# B&R Automation Studio project Parker_BMM_ST_V5_3147_V12 (part 13)

#### pullbottom.c
```c
/********************************************************************
 * COPYRIGHT --  B&R
 ********************************************************************
 * Program: bullbottom
 * File: pullbottom.c
 * Author: lijianjun
 * Created: March 06, 2013
 ********************************************************************
 * Implementation of program coolpin --- pull bottom control
 ********************************************************************/

#include <bur/plctypes.h>

#ifdef _DEFAULT_INCLUDES
	#include <AsDefault.h>
#endif

/**************************************************************************************
                            Function Declarations
**************************************************************************************/

void PullBottom( Mold_typ * pMold);

/**************************************************************************************
     	        		I N I T U P  O F   T H E   T A S K
**************************************************************************************/
_INIT void init ( void )
 {
	LMold.PullBottom.Step = 0;
 	RMold.PullBottom.Step = 0;
 } /* end of _INIT */

 /*************************************************************************************
        				C Y C L I C   P A R T   O F   T H E   T A S K
**************************************************************************************/

 _CYCLIC void cyclic ( void )
 {

	PullBottom(&LMold);
	PullBottom(&RMold);

	gMachineOut.LMold.PullBottom = LMold.ValveOut.PullBottom;
	gMachineOut.RMold.PullBottom = RMold.ValveOut.PullBottom;

 } /* end of _CYCLIC */

void PullBottom( Mold_typ * pMold)
{
   if(0 == pMold->TimeSet.CoolPinUpAlarmTime)pMold->TimeSet.CoolPinUpAlarmTime = 500;

   switch ( pMold->PullBottom.Step )
   {
         /*------------------ stop all the output ------------------*/
         case 0:
            pMold->ValveOut.PullBottom  = 0;
            pMold->ActInfo.PullBottom   = 0;
			pMold->PullBottom.Timer.IN	   = 0;
            break;

      	/*------------------ PullBottom -------------------- */
         case 100: /* PullBottom delay*/
            if(pMold->Option.PullBottom)
            {
				if(pMold->TimeSet.PullBottomDelay != 0)
				{
					pMold->PullBottom.Timer.IN = 1;
					pMold->PullBottom.Timer.PT = pMold->TimeSet.PullBottomDelay;
					pMold->PullBottom.Step = 200;
				}
				else
				{
					pMold->PullBottom.Step = 300;
				}

            }
            else
            {
            	pMold->PullBottom.Step = 900;
            }
          	break;

         case 200: /* delay ok */
            pMold->TimeDis.PullBottomDelay = pMold->PullBottom.Timer.ET;
            if (1 == pMold->PullBottom.Timer.Q)
            {
               pMold->PullBottom.Timer.IN       = 0;
               pMold->TimeDis.CoolPinDnDelay = 0;
               pMold->PullBottom.Step = 300;
            }
            break;

         case 300:

            if(pMold->TimeSet.PullBottomTime != 0)
            {
               pMold->PullBottom.Timer.IN = 1;
               pMold->PullBottom.Timer.PT = pMold->TimeSet.PullBottomTime;
               pMold->PullBottom.Step = 400;
            }
            else
            {
               pMold->PullBottom.Step = 500;
            }
            break;

         case 400: /*PullBottom time*/
            pMold->ActInfo.PullBottom  = 1;
            pMold->ValveOut.PullBottom = 1;

            pMold->TimeDis.PullBottomTime = pMold->PullBottom.Timer.ET;
            if (1 == pMold->PullBottom.Timer.Q)
            {
               pMold->ValveOut.PullBottom = 0;
               pMold->PullBottom.Timer.IN = 0;
//               pMold->TimeDis.PullBottomTime = 0;
               pMold->PullBottom.Step = 500;
            }

            break;

		case 500:
			pMold->ActInfo.PullBottom  = 0;
			pMold->ValveOut.PullBottom = 0;

			pMold->PullBottom.Step = 900;

			break;

         case 900:

			pMold->ActInfo.PullBottom  = 0;
			pMold->ValveOut.PullBottom = 0;

			pMold->PullBottom.Timer.IN = 0;

			pMold->PullBottom.Step = 3000;

            break;

		case 1100:      /* bCoolPinUpNextCycClampCls  autorun Case-4570 */
						/* 強制桿下到下一循環關模後才轉一上 */

			pMold->ActInfo.CoolPinDn  = 1;
			pMold->ValveOut.CoolPinDn = 1;

			break;

         case 3000:
            break;

		case 5000:
			pMold->ActInfo.PullBottom  = 1;
			pMold->ValveOut.PullBottom = 1;

			break;

         case 20000:
            pMold->ActInfo.PullBottom  = 0;
            pMold->ValveOut.PullBottom = 0;

			pMold->PullBottom.Timer.IN = 0;
            pMold->PullBottom.Step = 0;
            break;

		case 30000:
			pMold->ActInfo.PullBottom  = 0;
			pMold->ValveOut.PullBottom = 0;

			pMold->PullBottom.Timer.IN = 0;
			pMold->PullBottom.Step = 0;
            break;

   }/* end of switch */

	/* ----------------- pull bottom  action limit --------------------  */
	if(pMold->PullBottom.Step > 100 && pMold->PullBottom.Step < 900)
	{

	}

}/*end of function */
```

### Program Logical/process/hookpin (ANSIC, version 1.00.0) - hook pin

#### hookpin.c
```c
/********************************************************************
 * COPYRIGHT --  B&R
 ********************************************************************
 * Program: HookPin
 * File: HookPin.c
 * Author: lijianjun
 * Created: March 06, 2013
 ********************************************************************
 * Implementation of program HookPin --- cooling pin control
 ********************************************************************/

#include <bur/plctypes.h>

#ifdef _DEFAULT_INCLUDES
#include <AsDefault.h>
#endif

/**************************************************************************************
                            Function Declarations
**************************************************************************************/

void HookPin( Mold_typ * pMold);

/**************************************************************************************
     	        		I N I T U P  O F   T H E   T A S K
**************************************************************************************/
_INIT void init ( void )
{
	LMold.HookPin.Step = 0;
	RMold.HookPin.Step = 0;
} /* end of _INIT */

 /*************************************************************************************
        				C Y C L I C   P A R T   O F   T H E   T A S K
**************************************************************************************/

_CYCLIC void cyclic ( void )
{

	LMold.TransDIn.HookPinFwLimit = gMachineIn.LMold.HookPinFwLimit;
	RMold.TransDIn.HookPinFwLimit = gMachineIn.RMold.HookPinFwLimit;

	LMold.TransDIn.HookPinBwLimit = gMachineIn.LMold.HookPinBwLimit;
	RMold.TransDIn.HookPinBwLimit = gMachineIn.RMold.HookPinBwLimit;

	HookPin(&LMold);
	HookPin(&RMold);

	gMachineOut.LMold.HookPinFw = LMold.ValveOut.HookPinFw;
	gMachineOut.RMold.HookPinFw = RMold.ValveOut.HookPinFw;

} /* end of _CYCLIC */

void HookPin( Mold_typ * pMold)
{
	if(0 == pMold->TimeSet.HookPinFwAlarmTime)pMold->TimeSet.HookPinFwAlarmTime = 500;
	if(0 == pMold->TimeSet.HookPinBwAlarmTime)pMold->TimeSet.HookPinBwAlarmTime = 500;

	switch ( pMold->HookPin.Step )
	{
		/*------------------ stop all the output ------------------*/
		case 0:
//			pMold->ActInfo.HookPinFw   = 0;
//			pMold->ValveOut.HookPinFw  = 0;

			pMold->HookPin.LimitTimer.IN	   = 0;
			pMold->HookPin.Timer.IN	   = 0;
			break;

		/*--------------------------------------------------- */
		/*---------------- HookPin Fw  --------------------- */
		/*--------------------------------------------------- */
		case 100: /* HookPin delay*/
			if(pMold->Option.HookPin)
			{
				if(pMold->TimeSet.HookPinFwDelay != 0)
				{
					pMold->HookPin.Timer.IN = 1;
					pMold->HookPin.Timer.PT = pMold->TimeSet.HookPinFwDelay;
					pMold->HookPin.Step = 200;
				}
				else
				{
					pMold->HookPin.Step = 300;
				}
			}
			else
			{
				pMold->HookPin.Step = 300;
			}
			break;

		case 200: /* delay ok */
			pMold->TimeDis.HookPinFwDelay = pMold->HookPin.Timer.ET;
			if (1 == pMold->HookPin.Timer.Q)
			{
				pMold->HookPin.Timer.IN       = 0;
				//               pMold->TimeDis.HookPinFwDelay = 0;
				pMold->HookPin.Step = 300;
			}
			break;

		case 300:
			if(pMold->Option.HookPin)
			{
				pMold->HookPin.LimitTimer.IN = 1;
				pMold->HookPin.LimitTimer.PT = pMold->TimeSet.HookPinFwAlarmTime;
				pMold->HookPin.Step = 400;
			}
			else
			{
				pMold->HookPin.Step = 2900;  // for no use
			}

			break;

		case 400:
			pMold->ActInfo.HookPinFw  = 1;
			pMold->ValveOut.HookPinFw = 1;

			if (1 == pMold->TransDIn.HookPinFwLimit)
			{
				pMold->HookPin.Step = 500;
			}

			break;

		case 500:

			pMold->HookPin.LimitTimer.IN	   = 0;
			pMold->HookPin.Timer.IN	   = 0;

			pMold->HookPin.Step = 3000;
			break;

		case 2900:  // for no use

			pMold->ActInfo.HookPinFw   = 0;
			pMold->ValveOut.HookPinFw  = 0;

			pMold->HookPin.LimitTimer.IN	   = 0;
			pMold->HookPin.Timer.IN	   = 0;

			pMold->HookPin.Step = 3000;

			break;

		case 3000:
			break;

		case 5000:
			pMold->ActInfo.HookPinFw  = 1;
			pMold->ValveOut.HookPinFw = 1;

			break;

		/*--------------------------------------------------- */
		/*---------------- HookPin Bw  --------------------- */
		/*--------------------------------------------------- */

		case 10100: /* HookPin delay*/
			if(pMold->Option.HookPin)
			{
				if(pMold->TimeSet.HookPinBwDelay != 0)
				{
					pMold->HookPin.Timer.IN = 1;
					pMold->HookPin.Timer.PT = pMold->TimeSet.HookPinBwDelay;
					pMold->HookPin.Step = 10200;
				}
				else
				{
					pMold->HookPin.Step = 10300;
				}
			}
			else
			{
				pMold->HookPin.Step = 10300;
			}
			break;

		case 10200: /* delay ok */
			pMold->TimeDis.HookPinBwDelay = pMold->HookPin.Timer.ET;
			if (1 == pMold->HookPin.Timer.Q)
			{
				pMold->HookPin.Timer.IN       = 0;
				//               pMold->TimeDis.HookPinFwDelay = 0;
				pMold->HookPin.Step = 10300;
			}
			break;

		case 10300:

			if(pMold->Option.HookPin)
			{
				pMold->HookPin.LimitTimer.IN = 1;
				pMold->HookPin.LimitTimer.PT = pMold->TimeSet.HookPinBwAlarmTime;
				pMold->HookPin.Step = 10400;
			}
			else
			{

				if (1 == pMold->TransDIn.HookPinBwLimit)
				{
					pMold->HookPin.Step = 12900;  // for no use
				}
				else
				{
					pMold->Alarm.HookPinNotAtBwPos = 1;
					pMold->HookPin.Step = 40000;           /*  HookPin bw alarm   */
				}
			}

			break;

		case 10400:

			pMold->ActInfo.HookPinFw  = 0;
			pMold->ValveOut.HookPinFw = 0;

			if (1 == pMold->TransDIn.HookPinBwLimit)
			{
				pMold->HookPin.Step = 10500;
			}

			break;

		case 10500:

			pMold->ActInfo.HookPinFw   = 0;
			//			pMold->ValveOut.HookPinFw  = 0;

			pMold->HookPin.LimitTimer.IN	   = 0;
			pMold->HookPin.Timer.IN	   = 0;

			pMold->HookPin.Step = 13000;

			break;

		case 12900:  // for no use

			pMold->ActInfo.HookPinFw   = 0;
			pMold->ValveOut.HookPinFw  = 0;

			pMold->HookPin.LimitTimer.IN	   = 0;
			pMold->HookPin.Timer.IN	   = 0;

			pMold->HookPin.Step = 13000;

			break;

		case 13000:

			break;

		case 15000:
			pMold->ActInfo.HookPinFw  = 0;
			pMold->ValveOut.HookPinFw = 0;

			break;

		case 20000:
//			pMold->ActInfo.HookPinFw   = 0;
//			pMold->ValveOut.HookPinFw  = 0;

			pMold->HookPin.LimitTimer.IN	   = 0;
			pMold->HookPin.Timer.IN	   = 0;

			pMold->HookPin.Step	   = 0;
			break;

		case 30000:
			//			pMold->ActInfo.HookPinFw   = 0;
			//			pMold->ValveOut.HookPinFw  = 0;

			pMold->HookPin.LimitTimer.IN	   = 0;
			pMold->HookPin.Timer.IN	   = 0;

			pMold->HookPin.Step	   = 0;
			break;

		case 40000:
			//			pMold->ActInfo.HookPinFw   = 0;
			//			pMold->ValveOut.HookPinFw  = 0;

			pMold->HookPin.LimitTimer.IN	   = 0;
			pMold->HookPin.Timer.IN	   = 0;

			break;

		case 41000:
			//			pMold->ActInfo.HookPinFw   = 0;
			//			pMold->ValveOut.HookPinFw  = 0;

			pMold->HookPin.LimitTimer.IN	   = 0;
			pMold->HookPin.Timer.IN	   = 0;

			pMold->HookPin.Step	   = 40000;

			break;
	}/* end of switch */

	/* ----------------- HookPin Fw / Bw timeout --------------------  */
	if(1 == pMold->HookPin.LimitTimer.Q && 1 == gMachineInfo.TimeLimit)
	{
		if(pMold->HookPin.Step < 500 && pMold->HookPin.Step > 300)		/* HookPin Fw  */
		{
			pMold->Alarm.HookPinNotAtFwPos = 1;
		}

		if(pMold->TopDeflash.Step < 10500 && pMold->TopDeflash.Step > 10300)	/* HookPin Bw  */
		{
			pMold->Alarm.HookPinNotAtBwPos = 1;
		}

		pMold->HookPin.Step = 41000;
	}

	/* ----------------- Angle pin Fw  action limit --------------------  */
	if(pMold->HookPin.Step > 300 && pMold->HookPin.Step < 500)
	{
		if( 0 == pMold->Carriage.BwPos )
		{
			pMold->Alarm.CarriageNotAtBwDI= 1;
			pMold->HookPin.Step = 40000;
		}
	}

}/*end of function */
```

### Program Logical/process/coolpin (ANSIC, version 1.00.0) - cool pin

#### coolpin.c
```c
/********************************************************************
 * COPYRIGHT --  B&R
 ********************************************************************
 * Program: coolpin
 * File: coolpin.c
 * Author: lijianjun
 * Created: March 06, 2013
 ********************************************************************
 * Implementation of program coolpin --- cooling pin control
 ********************************************************************/

#include <bur/plctypes.h>

#ifdef _DEFAULT_INCLUDES
#include <AsDefault.h>
#endif

/**************************************************************************************
                            Function Declarations
**************************************************************************************/

void CoolPin( Mold_typ * pMold);

/**************************************************************************************
     	        		I N I T U P  O F   T H E   T A S K
**************************************************************************************/
_INIT void init ( void )
{
	LMold.CoolPin.Step = 0;
	RMold.CoolPin.Step = 0;
} /* end of _INIT */

 /*************************************************************************************
        				C Y C L I C   P A R T   O F   T H E   T A S K
**************************************************************************************/

_CYCLIC void cyclic ( void )
{

	LMold.TransDIn.CoolPinUpLimit = gMachineIn.LMold.CoolPinUpLimit;
	RMold.TransDIn.CoolPinUpLimit = gMachineIn.RMold.CoolPinUpLimit;

	CoolPin(&LMold);
	CoolPin(&RMold);

	gMachineOut.LMold.CoolPinDn = LMold.ValveOut.CoolPinDn;
	gMachineOut.RMold.CoolPinDn = RMold.ValveOut.CoolPinDn;

} /* end of _CYCLIC */

void CoolPin( Mold_typ * pMold)
{
	if(0 == pMold->TimeSet.CoolPinUpAlarmTime)pMold->TimeSet.CoolPinUpAlarmTime = 500;

	switch ( pMold->CoolPin.Step )
	{
		/*------------------ stop all the output ------------------*/
		case 0:
//			pMold->ValveOut.CoolPinDn  = 0;
//			pMold->ActInfo.CoolPinDn   = 0;
			pMold->CoolPin.LimitTimer.IN	   = 0;
			pMold->CoolPin.Timer.IN	   = 0;
			break;

		/*------------------ CoolPin -------------------- */
		case 100: /* CoolPin delay*/
			if(pMold->Option.CoolPin)
			{
				if ( 1 == gMachineFix.Option.bCoolPinUpNextCycClampCls)    /*  於下一循環關模後轉一上    */
				{
					pMold->CoolPin.Step = 1100; 		/*  強制桿下到下一循環關模後才轉一上 */
				}
				else
				{
					if(pMold->TimeSet.CoolPinDnDelay != 0)
					{
						pMold->CoolPin.Timer.IN = 1;
						pMold->CoolPin.Timer.PT = pMold->TimeSet.CoolPinDnDelay;
						pMold->CoolPin.Step = 200;

						//gExSPC
						if(pMold == & LMold)
						{
							gExSPC[ExIndex].LMold.CoolPinDnDelay = pMold->TimeSet.CoolPinDnDelay/100.0;
						}
						else
						{
							gExSPC[ExIndex].RMold.CoolPinDnDelay = pMold->TimeSet.CoolPinDnDelay/100.0;
						}
					}
					else
					{
						pMold->CoolPin.Step = 300;
					}
				}
			}
			else
			{
				pMold->CoolPin.Step = 900;
			}
			break;

		case 200: /* delay ok */
			pMold->TimeDis.CoolPinDnDelay = pMold->CoolPin.Timer.ET;
			if (1 == pMold->CoolPin.Timer.Q)
			{
				pMold->CoolPin.Timer.IN       = 0;
				//               pMold->TimeDis.CoolPinDnDelay = 0;
				pMold->CoolPin.Step = 300;
			}
			break;

		case 300: //沒有轉一下時間， 轉一下直到轉一吹冷結束

			//            if(pMold->TimeSet.CoolPinDnTime != 0)
			//            {
			//               pMold->CoolPin.Timer.IN = 1;
			//               pMold->CoolPin.Timer.PT = pMold->TimeSet.CoolPinDnTime;
			//               pMold->CoolPin.Step = 400;
			//
			//				//gExSPC
			//				if(pMold == & LMold)
			//				{
			//					gExSPC[ExIndex].LMold.CoolPinDnTime = pMold->TimeSet.CoolPinDnTime/100.0;
			//				}
			//				else
			//				{
			//					gExSPC[ExIndex].RMold.CoolPinDnTime = pMold->TimeSet.CoolPinDnTime/100.0;
			//				}
			//            }
			//            else
			//            {
			//               pMold->CoolPin.Step = 500;
			//            }

			pMold->CoolPin.Step = 400;
			break;

		case 400:
			pMold->ActInfo.CoolPinDn  = 1;
			pMold->ValveOut.CoolPinDn = 1;

			//            pMold->TimeDis.CoolPinDnTime = pMold->CoolPin.Timer.ET;
			//            if (1 == pMold->CoolPin.Timer.Q)
			//            {
			//               pMold->ValveOut.CoolPinDn = 0;
			//               pMold->CoolPin.Timer.IN = 0;
			//               pMold->TimeDis.CoolPinDnTime = 0;
			//               pMold->CoolPin.Step = 500;
			//            }

			if (3000==pMold->CoolPinBlow.Step)
			{
				pMold->CoolPin.Step = 500;
			}

			break;

		case 500:

			if ((1 == pMold->Option.CoolPin) || (1 == pMold->ValveOut.CoolPinDn))
			{
				pMold->CoolPin.LimitTimer.IN = 1;
				pMold->CoolPin.LimitTimer.PT = pMold->TimeSet.CoolPinUpAlarmTime;
				pMold->CoolPin.Step = 600;
			}
			else
			{
				pMold->CoolPin.Step = 650;	// for no use
			}

			break;

		case 600:
			pMold->ActInfo.CoolPinDn  = 0;
			pMold->ValveOut.CoolPinDn = 0;

			if(pMold->TransDIn.CoolPinUpLimit)
			{
				pMold->CoolPin.Step = 900;
			}
			pMold->TimeDis.CoolPinUpAlarmTime = pMold->CoolPin.LimitTimer.ET;
			if (1 == pMold->CoolPin.LimitTimer.Q)
			{
				pMold->ActInfo.CoolPinDn  = 0;
				pMold->ValveOut.CoolPinDn = 0;

				pMold->CoolPin.LimitTimer.IN = 0;
				pMold->Alarm.CoolPinNotAtUpPos = 1;

				pMold->CoolPin.Step = 40000;
			}
			break;

		case 650: // for no use
			//			pMold->ActInfo.CoolPinDn  = 0;
			//			pMold->ValveOut.CoolPinDn = 0;

			if(pMold->TransDIn.CoolPinUpLimit)
			{
				pMold->CoolPin.Step = 900;
			}
			else
			{
				pMold->CoolPin.LimitTimer.IN = 0;
				pMold->Alarm.CoolPinNotAtUpPos = 1;

				pMold->CoolPin.Step = 40000;
			}

			//			pMold->TimeDis.CoolPinUpAlarmTime = pMold->CoolPin.LimitTimer.ET;
			//			if (1 == pMold->CoolPin.LimitTimer.Q)
			//			{
			//				pMold->CoolPin.LimitTimer.IN = 0;
			//				pMold->Alarm.CoolPinNotAtUpPos = 1;
			//
			//				pMold->CoolPin.Step = 40000;
			//			}
			break;

		case 900:

			pMold->ValveOut.CoolPinDn = 0;
			pMold->ActInfo.CoolPinDn  = 0;
			pMold->CoolPin.LimitTimer.IN = 0;
			pMold->CoolPin.Step = 3000;
			break;

		case 1100:      /* bCoolPinUpNextCycClampCls  autorun Case-4570 */
			/* 強制桿下到下一循環關模後才轉一上 */

			pMold->ActInfo.CoolPinDn  = 1;
			pMold->ValveOut.CoolPinDn = 1;

			break;

		case 3000:
			break;

		case 5000:
			pMold->ActInfo.CoolPinDn  = 1;
			pMold->ValveOut.CoolPinDn = 1;

			break;

		case 15000:
			pMold->ActInfo.CoolPinDn  = 0;
			pMold->ValveOut.CoolPinDn = 0;

			break;

		case 20000:
//			pMold->ActInfo.CoolPinDn  = 0;
//			pMold->ValveOut.CoolPinDn = 0;

			pMold->CoolPin.Timer.IN = 0;
			pMold->CoolPin.LimitTimer.IN = 0;
			pMold->CoolPin.Step = 0;
			break;

		case 30000:
//			pMold->ActInfo.CoolPinDn  = 0;
//			pMold->ValveOut.CoolPinDn = 0;
			pMold->CoolPin.Timer.IN = 0;
			pMold->CoolPin.LimitTimer.IN = 0;
			pMold->CoolPin.Step = 0;
			break;

		case 40000:
//			pMold->ActInfo.CoolPinDn  = 0;
//			pMold->ValveOut.CoolPinDn = 0;
			pMold->CoolPin.Timer.IN = 0;
			pMold->CoolPin.LimitTimer.IN = 0;

			break;
	}/* end of switch */

	/* ----------------- cool pin down  action limit --------------------  */
	if(pMold->CoolPin.Step > 100 && pMold->CoolPin.Step < 900)
	{

	}

}/*end of function */
```

### Program Logical/process/coolpin2 (ANSIC, version 1.00.0) - cool pin 2

#### coolpin2.c
```c
/********************************************************************
 * COPYRIGHT --  B&R
 ********************************************************************
 * Program: coolpin2
 * File: coolpin2.c
 * Author: lijianjun
 * Created: March 06, 2013
 ********************************************************************
 * Implementation of program coolpin2 --- cooling pin 2 control
 ********************************************************************/

#include <bur/plctypes.h>

#ifdef _DEFAULT_INCLUDES
	#include <AsDefault.h>
#endif

/**************************************************************************************
                            Function Declarations
**************************************************************************************/

void CoolPin2( Mold_typ * pMold);

/**************************************************************************************
     	        		I N I T U P  O F   T H E   T A S K
**************************************************************************************/
_INIT void init ( void )
 {
 	LMold.CoolPin2.Step = 0;
 	RMold.CoolPin2.Step = 0;
 } /* end of _INIT */

 /*************************************************************************************
        				C Y C L I C   P A R T   O F   T H E   T A S K
**************************************************************************************/

 _CYCLIC void cyclic ( void )
 {
 	LMold.TransDIn.CoolPin2UpLimit = gMachineIn.LMold.CoolPin2UpLimit;
 	RMold.TransDIn.CoolPin2UpLimit = gMachineIn.RMold.CoolPin2UpLimit;

	CoolPin2(&LMold);
	CoolPin2(&RMold);

	gMachineOut.LMold.CoolPin2Dn = LMold.ValveOut.CoolPin2Dn;
	gMachineOut.RMold.CoolPin2Dn = RMold.ValveOut.CoolPin2Dn;

 } /* end of _CYCLIC */

void CoolPin2( Mold_typ * pMold)
{
	if(0 == pMold->TimeSet.CoolPin2UpAlarmTime)pMold->TimeSet.CoolPin2UpAlarmTime = 500;

	switch ( pMold->CoolPin2.Step )
	{
		/*------------------ stop all the output ------------------*/
		case 0:
//			pMold->CoolPin2.Out   	   = 0;
//			pMold->ValveOut.CoolPin2Dn  = 0;
//			pMold->ActInfo.CoolPin2Dn   = 0;
			pMold->CoolPin2.Timer.IN	   = 0;
			pMold->CoolPin2.LimitTimer.IN	   = 0;
			break;

		/*------------------ CoolPin2 -------------------- */
		case 100: /* CoolPin2 delay*/
			if(pMold->Option.CoolPin2)
			{
				if(pMold->TimeSet.CoolPin2DnDelay != 0)
				{
					pMold->CoolPin2.Timer.IN = 1;
					pMold->CoolPin2.Timer.PT = pMold->TimeSet.CoolPin2DnDelay;
					pMold->CoolPin2.Step = 200;
				}
				else
				{
					pMold->CoolPin2.Step = 300;
				}
			}
			else
			{
				pMold->CoolPin2.Step = 500;
			}

			break;
		case 200: /* delay ok */
			pMold->TimeDis.CoolPin2DnDelay = pMold->CoolPin2.Timer.ET;
			if (1 == pMold->CoolPin2.Timer.Q)
			{
				pMold->CoolPin2.Timer.IN       = 0;
				//		pMold->TimeDis.CoolPin2DnDelay = 0;
				pMold->CoolPin2.Step = 400;
			}
			break;

		case 300:  //沒有轉二下時間， 轉二下直到轉二吹冷結束
			//            	if(pMold->TimeSet.CoolPin2DnTime != 0)
			//            	{
			//            		pMold->CoolPin2.Timer.IN = 1;
			//					pMold->CoolPin2.Timer.PT = pMold->TimeSet.CoolPin2DnTime;
			//					pMold->CoolPin2.Step = 400;
			//            	}
			//            	else
			//            	{
			//            		pMold->CoolPin2.Step = 500;
			//            	}
			pMold->CoolPin2.Step = 400;
			break;

		case 400:
			pMold->ActInfo.CoolPin2Dn  = 1;
			pMold->ValveOut.CoolPin2Dn = 1;
			pMold->CoolPin2.Out        = 1;

			//            	pMold->TimeDis.CoolPin2DnTime = pMold->CoolPin2.Timer.ET;
			//            	if (1 == pMold->CoolPin2.Timer.Q)
			//            	{
			//            		pMold->CoolPin2.Out        = 0;
			//            		pMold->ValveOut.CoolPin2Dn = 0;
			//            		pMold->CoolPin2.Timer.IN = 0;
			//            		pMold->TimeDis.CoolPin2DnTime = 0;
			//            		pMold->CoolPin2.Step = 500;
			//            	}
			if (3000==pMold->CoolPin2Blow.Step)
			{
				pMold->CoolPin2.Step = 500;
			}

			break;

		case 500:
			pMold->CoolPin2.Timer.IN = 0;
			pMold->CoolPin2.Step = 550;
			break;

		case 550:
			if (1 == pMold->Option.CoolPin2)
			{
				pMold->CoolPin2.LimitTimer.IN = 1;
				pMold->CoolPin2.LimitTimer.PT = pMold->TimeSet.CoolPin2UpAlarmTime;
				pMold->CoolPin2.Step = 600;
			}
			else
			{
				pMold->CoolPin2.Step = 650;	// for no use
			}

			break;

		case 600:
			pMold->ActInfo.CoolPin2Dn  = 0;
			pMold->CoolPin2.Out        = 0;
			pMold->ValveOut.CoolPin2Dn = 0;

			if(1 == pMold->TransDIn.CoolPin2UpLimit)
			{
				pMold->CoolPin2.Step = 900;
			}
			pMold->TimeDis.CoolPin2UpAlarmTime = pMold->CoolPin2.LimitTimer.ET;

			if (1 == pMold->CoolPin2.LimitTimer.Q)
			{
				pMold->ActInfo.CoolPin2Dn  = 0;
				pMold->CoolPin2.Out        = 0;
				pMold->ValveOut.CoolPin2Dn = 0;

				pMold->CoolPin2.LimitTimer.IN = 0;
				pMold->Alarm.CoolPin2NotAtUpPos = 1;

				pMold->CoolPin2.Step = 40000;
			}
			break;

		case 650: // for no use

			if(pMold->TransDIn.CoolPin2UpLimit)
			{
				pMold->CoolPin2.Step = 900;
			}
			else
			{
				pMold->CoolPin2.LimitTimer.IN = 0;
				pMold->Alarm.CoolPin2NotAtUpPos = 1;
				pMold->CoolPin2.Step = 40000;
			}

			//			pMold->TimeDis.CoolPin2UpAlarmTime = pMold->CoolPin2.Timer.ET;
			//			if (1 == pMold->CoolPin2.Timer.Q)
			//			{
			//			//	pMold->ActInfo.CoolPin2Dn  = 0;
			//			//	pMold->CoolPin2.Out        = 0;
			//			//	pMold->ValveOut.CoolPin2Dn = 0;
			//
			//				pMold->CoolPin2.Timer.IN = 0;
			//				pMold->Alarm.CoolPin2NotAtUpPos = 1;
			//
			//				pMold->CoolPin2.Step = 40000;
			//			}
			break;

		case 900:
			if (1==gMachineInfo.Auto)
			{
				if(pMold == &RMold)
				{
					RMold.Option.CoolPin2 = gMacOption.RCoolPin2;
				}
				else
				{
					LMold.Option.CoolPin2 = gMacOption.LCoolPin2;
				}
			}
			pMold->CoolPin2.Out      = 0;
			pMold->ValveOut.CoolPin2Dn  = 0;
			pMold->ActInfo.CoolPin2Dn   = 0;

			pMold->CoolPin2.Timer.IN = 0;
			pMold->CoolPin2.LimitTimer.IN = 0;
			pMold->CoolPin2.Step = 3000;
			break;
		case 3000:

			break;

		case 5000:
			pMold->ActInfo.CoolPin2Dn  = 1;
			pMold->ValveOut.CoolPin2Dn = 1;

			break;

		case 15000:
			pMold->ActInfo.CoolPin2Dn  = 0;
			pMold->ValveOut.CoolPin2Dn = 0;

			break;

		case 20000:
//			pMold->CoolPin2.Out        = 0;
//			pMold->ActInfo.CoolPin2Dn  = 0;
//			pMold->ValveOut.CoolPin2Dn = 0;

			pMold->CoolPin2.Timer.IN = 0;
			pMold->CoolPin2.LimitTimer.IN = 0;
			pMold->CoolPin2.Step    = 0;
			break;

		case 30000:
//			pMold->CoolPin2.Out        = 0;
//			pMold->ActInfo.CoolPin2Dn  = 0;
//			pMold->ValveOut.CoolPin2Dn = 0;
			pMold->CoolPin2.Timer.IN = 0;
			pMold->CoolPin2.LimitTimer.IN = 0;
			pMold->CoolPin2.Step     = 0;
			break;

		case 40000:
//			pMold->CoolPin2.Out        = 0;
//			pMold->ActInfo.CoolPin2Dn  = 0;
//			pMold->ValveOut.CoolPin2Dn = 0;
			pMold->CoolPin2.Timer.IN = 0;
			pMold->CoolPin2.LimitTimer.IN = 0;

			break;

		case 41000:
			//			pMold->CoolPin2.Out        = 0;
			//			pMold->ActInfo.CoolPin2Dn  = 0;
			//			pMold->ValveOut.CoolPin2Dn = 0;
			pMold->CoolPin2.Timer.IN = 0;
			pMold->CoolPin2.LimitTimer.IN = 0;
			pMold->CoolPin2.Step     = 40000;
			break;

	}/* end of switch */

	/* ----------------- cool pin2 down  action limit --------------------  */
	if(pMold->CoolPin2.Step > 100 && pMold->CoolPin2.Step < 900)
	{

	}

}/*end of function */
```

### Program Logical/process/coolpin3 (ANSIC, version 1.00.0) - cool pin 3

#### coolpin3.c
```c
/********************************************************************
 * COPYRIGHT --  B&R
 ********************************************************************
 * Program: coolpin3
 * File: coolpin3.c
 * Author: lijianjun
 * Created: March 06, 2013
 ********************************************************************
 * Implementation of program coolpin3 --- cooling pin 3 control
 ********************************************************************/

#include <bur/plctypes.h>

#ifdef _DEFAULT_INCLUDES
#include <AsDefault.h>
#endif

/**************************************************************************************
                            Function Declarations
**************************************************************************************/

void CoolPin3( Mold_typ * pMold);

/**************************************************************************************
     	        		I N I T U P  O F   T H E   T A S K
**************************************************************************************/
_INIT void init ( void )
{
	LMold.CoolPin3.Step = 0;
	RMold.CoolPin3.Step = 0;
} /* end of _INIT */

 /*************************************************************************************
        				C Y C L I C   P A R T   O F   T H E   T A S K
**************************************************************************************/

_CYCLIC void cyclic ( void )
{
	LMold.TransDIn.CoolPin3UpLimit = gMachineIn.LMold.CoolPin3UpLimit;
	RMold.TransDIn.CoolPin3UpLimit = gMachineIn.RMold.CoolPin3UpLimit;

	CoolPin3(&LMold);
	CoolPin3(&RMold);

	gMachineOut.LMold.CoolPin3Dn = LMold.ValveOut.CoolPin3Dn;
	gMachineOut.RMold.CoolPin3Dn = RMold.ValveOut.CoolPin3Dn;

} /* end of _CYCLIC */

void CoolPin3( Mold_typ * pMold)
{

	if(0 == pMold->TimeSet.CoolPin3UpAlarmTime)pMold->TimeSet.CoolPin3UpAlarmTime = 500;

	switch ( pMold->CoolPin3.Step )
	{
		/*------------------ stop all the output ------------------*/
		case 0:
//			pMold->ActInfo.CoolPin3Dn   = 0;
//			pMold->ValveOut.CoolPin3Dn  = 0;

			pMold->CoolPin3.LimitTimer.IN = 0;
			pMold->CoolPin3.Timer.IN	= 0;
			break;

		/*------------------ CoolPin3 -------------------- */
		case 100: /* CoolPin3 delay*/
			if(pMold->Option.CoolPin3)
			{
				if(pMold->TimeSet.CoolPin3DnDelay != 0)
				{
					pMold->CoolPin3.Timer.IN = 1;
					pMold->CoolPin3.Timer.PT = pMold->TimeSet.CoolPin3DnDelay;
					pMold->CoolPin3.Step = 200;
				}
				else
				{
					pMold->CoolPin3.Step = 400;
				}
			}
			else
			{
				pMold->CoolPin3.Step = 900;
			}
			break;
		case 200: /* delay ok */
			pMold->TimeDis.CoolPin3DnDelay = pMold->CoolPin3.Timer.ET;
			if (1 == pMold->CoolPin3.Timer.Q)
			{
				pMold->CoolPin3.Timer.IN       = 0;
				//	pMold->TimeDis.CoolPin3DnDelay = 0;
				pMold->CoolPin3.Step = 400;
			}
			break;
		case 300:  //沒有轉三下時間， 轉三下直到轉三吹冷結束
			//            	if(pMold->TimeSet.CoolPin3DnTime != 0)
			//            	{
			//            		pMold->CoolPin3.Timer.IN = 1;
			//					pMold->CoolPin3.Timer.PT = pMold->TimeSet.CoolPin3DnTime;
			//					pMold->CoolPin3.Step = 400;
			//            	}
			//            	else
			//            	{
			//            		pMold->CoolPin3.Step = 500;
			//            	}
			pMold->CoolPin3.Step = 400;

			break;
		case 400:
			pMold->ActInfo.CoolPin3Dn  = 1;
			pMold->ValveOut.CoolPin3Dn = 1;

			//            	pMold->TimeDis.CoolPin3DnTime = pMold->CoolPin3.Timer.ET;
			//            	if (1 == pMold->CoolPin3.Timer.Q)
			//            	{
			//            		pMold->ValveOut.CoolPin3Dn = 0;
			//            		pMold->CoolPin3.Timer.IN = 0;
			//            		pMold->TimeDis.CoolPin3DnTime = 0;
			//            		pMold->CoolPin3.Step = 450;
			//            	}
			if (3000==pMold->CoolPin3Blow.Step)
			{
				pMold->CoolPin3.Step = 500;
			}
			break;

		case 500:
			pMold->CoolPin3.Timer.IN = 0;
			pMold->CoolPin3.Step = 550;

			break;

		case 550:
			if (1 == pMold->Option.CoolPin3)
			{
				pMold->CoolPin3.LimitTimer.IN = 1;
				pMold->CoolPin3.LimitTimer.PT = pMold->TimeSet.CoolPin3UpAlarmTime;
				pMold->CoolPin3.Step = 600;
			}
			else
			{
				pMold->CoolPin3.Step = 650;	// for no use
			}

			break;

		case 600:
			pMold->ActInfo.CoolPin3Dn  = 0;
			pMold->ValveOut.CoolPin3Dn = 0;

			if(pMold->TransDIn.CoolPin3UpLimit)
			{
				pMold->CoolPin3.Step = 900;
			}
			pMold->TimeDis.CoolPin3UpAlarmTime = pMold->CoolPin3.LimitTimer.ET;
			if (1 == pMold->CoolPin3.LimitTimer.Q)
			{
				pMold->ActInfo.CoolPin3Dn  = 0;
				pMold->ValveOut.CoolPin3Dn = 0;

				pMold->CoolPin3.LimitTimer.IN = 0;
				pMold->Alarm.CoolPin3NotAtUpPos = 1;

				pMold->CoolPin3.Step = 40000;
			}
			break;

		case 650: // for no use

			if(pMold->TransDIn.CoolPin3UpLimit)
			{
				pMold->CoolPin3.Step = 900;
			}
			else
			{
				pMold->CoolPin3.LimitTimer.IN = 0;
				pMold->Alarm.CoolPin3NotAtUpPos = 1;
				pMold->CoolPin3.Step = 40000;
			}

			break;

		case 900:
			if (1==gMachineInfo.Auto)
			{
				if(pMold == &RMold)
				{
					RMold.Option.CoolPin3 = gMacOption.RCoolPin3;
				}
				else
				{
					LMold.Option.CoolPin3 = gMacOption.LCoolPin3;
				}
			}

			pMold->ValveOut.CoolPin3Dn  = 0;
			pMold->ActInfo.CoolPin3Dn   = 0;

			pMold->CoolPin3.Timer.IN = 0;
			pMold->CoolPin3.LimitTimer.IN = 0;
			pMold->CoolPin3.Step = 3000;

			break;

		case 3000:

			break;

		case 5000:
			pMold->ActInfo.CoolPin3Dn  = 1;
			pMold->ValveOut.CoolPin3Dn = 1;

			break;

		case 15000:
			pMold->ActInfo.CoolPin3Dn  = 0;
			pMold->ValveOut.CoolPin3Dn = 0;

			break;

		case 20000:
//			pMold->ActInfo.CoolPin3Dn  = 0;
//			pMold->ValveOut.CoolPin3Dn = 0;

			pMold->CoolPin3.Timer.IN = 0;
			pMold->CoolPin3.LimitTimer.IN = 0;
			pMold->CoolPin3.Step    = 0;
			break;

		case 30000:
//			pMold->ActInfo.CoolPin3Dn  = 0;
//			pMold->ValveOut.CoolPin3Dn = 0;

			pMold->CoolPin3.Timer.IN = 0;
			pMold->CoolPin3.LimitTimer.IN = 0;
			pMold->CoolPin3.Step     = 0;
			break;

		case 40000:
//			pMold->ActInfo.CoolPin3Dn  = 0;
//			pMold->ValveOut.CoolPin3Dn = 0;

			pMold->CoolPin3.Timer.IN = 0;
			pMold->CoolPin3.LimitTimer.IN = 0;

			break;

		case 41000:
			//			pMold->ActInfo.CoolPin3Dn  = 0;
			//			pMold->ValveOut.CoolPin3Dn = 0;

			pMold->CoolPin3.Timer.IN = 0;
			pMold->CoolPin3.LimitTimer.IN = 0;
			pMold->CoolPin3.Step     = 40000;
			break;

	}/* end of switch */

	/* ----------------- cool pin3 down  action limit --------------------  */
	if(pMold->CoolPin3.Step > 100 && pMold->CoolPin3.Step < 900)
	{

	}

}/*end of function */
```

### Program Logical/process/coolblw (ANSIC, version 1.00.0) - cooling blow

#### coolblow.c
```c
/********************************************************************
 * COPYRIGHT --  B&R
 ********************************************************************
 * Program: coolblow
 * File: coolblow.c
 * Author: lijianjun
 * Created: March 06, 2013
 ********************************************************************
 * Implementation of program coolblow --- cooling blow control
 ********************************************************************/

#include <bur/plctypes.h>
#ifdef _DEFAULT_INCLUDES
	#include <AsDefault.h>
#endif

/**************************************************************************************
                            Function Declarations
**************************************************************************************/

void CoolPinBlow( Mold_typ * pMold);

/**************************************************************************************
     	        		I N I T U P  O F   T H E   T A S K
**************************************************************************************/
_INIT void init ( void )
 {
 	LMold.CoolPinBlow.Step = 0;
 	RMold.CoolPinBlow.Step = 0;
 } /* end of _INIT */

 /*************************************************************************************
        				C Y C L I C   P A R T   O F   T H E   T A S K
**************************************************************************************/

 _CYCLIC void cyclic ( void )
 {
	CoolPinBlow(&LMold);
	CoolPinBlow(&RMold);

	gMachineOut.LMold.CoolPinBlow = LMold.ValveOut.CoolPinBlow;
	gMachineOut.RMold.CoolPinBlow = RMold.ValveOut.CoolPinBlow;

 } /* end of _CYCLIC */

void CoolPinBlow( Mold_typ * pMold)
{

	 switch ( pMold->CoolPinBlow.Step )
     {
      		/*------------------ stop all the output ------------------*/
            case 0:
            	pMold->ValveOut.CoolPinBlow   = 0;
            	pMold->ActInfo.CoolPinBlow  = 0;
            	pMold->CoolPinBlow.Timer.IN	= 0;
            	break;

      		/*------------------ CoolPin -------------------- */
            case 100:
            	if(pMold->Option.CoolPin)
      			{
	            	if(pMold->TimeSet.CoolPinBlowDelay != 0)
		      		{
	      				pMold->CoolPinBlow.Timer.IN = 1;
						pMold->CoolPinBlow.Timer.PT = pMold->TimeSet.CoolPinBlowDelay;
	      				pMold->CoolPinBlow.Step = 200;

						//gExSPC
						if(pMold == & LMold)
						{
							gExSPC[ExIndex].LMold.CoolPinBlowDelay = pMold->TimeSet.CoolPinBlowDelay/100.0;
						}
						else
						{
							gExSPC[ExIndex].RMold.CoolPinBlowDelay = pMold->TimeSet.CoolPinBlowDelay/100.0;
						}
	      			}
	      			else
	      			{
	      				pMold->CoolPinBlow.Step = 300;
	      			}
	      		}
	      		else
	      		{
	      			pMold->CoolPinBlow.Step = 900;
	      		}
            	break;
            case 200:
            	pMold->TimeDis.CoolPinBlowDelay = pMold->CoolPinBlow.Timer.ET;
            	if (1 == pMold->CoolPinBlow.Timer.Q)
            	{
            		pMold->CoolPinBlow.Timer.IN       = 0;
            	//	pMold->TimeDis.CoolPinBlowDelay = 0;
            		pMold->CoolPinBlow.Step = 300;
            	}
            	break;
            case 300:
            	if(pMold->TimeSet.CoolPinBlowTime != 0)
            	{
            		pMold->CoolPinBlow.Timer.IN = 1;
					pMold->CoolPinBlow.Timer.PT = pMold->TimeSet.CoolPinBlowTime;
					pMold->CoolPinBlow.Step = 400;

					//gExSPC
					if(pMold == & LMold)
					{
						gExSPC[ExIndex].LMold.CoolPinBlowTime = pMold->TimeSet.CoolPinBlowTime/100.0;
					}
					else
					{
						gExSPC[ExIndex].RMold.CoolPinBlowTime = pMold->TimeSet.CoolPinBlowTime/100.0;
					}

            	}
            	else
            	{
            		pMold->CoolPinBlow.Step = 900;
            	}
            	break;
            case 400:
            	pMold->ActInfo.CoolPinBlow  = 1;
            	pMold->ValveOut.CoolPinBlow = 1;

            	pMold->TimeDis.CoolPinBlowTime = pMold->CoolPinBlow.Timer.ET;
            	if (1 == pMold->CoolPinBlow.Timer.Q)
            	{
            		pMold->CoolPinBlow.Timer.IN = 0;
            	//	pMold->TimeDis.CoolPinBlowTime = 0;

            		pMold->CoolPinBlow.Step = 500;
            	}
            	break;

			case 500:
				pMold->ActInfo.CoolPinBlow  = 0;
				pMold->ValveOut.CoolPinBlow = 0;

				pMold->CoolPinBlow.Step = 900;

				break;

            case 900:
//			if (1==gMachineInfo.Auto)
//			{
//				if(pMold == &RMold)
//				{
//					RMold.Option.CoolPin = gMacOption.RCoolPin;
//				}
//				else
//				{
//					LMold.Option.CoolPin = gMacOption.LCoolPin;
//				}
//			}
            	pMold->ActInfo.CoolPinBlow  = 0;
            	pMold->ValveOut.CoolPinBlow = 0;

            	pMold->CoolPinBlow.Timer.IN = 0;

            	pMold->CoolPinBlow.Step = 3000;
            	break;

            case 3000:
            	break;

			case 5000:
				pMold->ActInfo.CoolPinBlow  = 1;
				pMold->ValveOut.CoolPinBlow = 1;

				break;

            case 20000:
            	pMold->ActInfo.CoolPinBlow  = 0;
            	pMold->ValveOut.CoolPinBlow = 0;

				pMold->CoolPinBlow.Timer.IN = 0;
				pMold->CoolPinBlow.Step    = 0;
				break;

			case 30000:
            	pMold->ActInfo.CoolPinBlow  = 0;
            	pMold->ValveOut.CoolPinBlow = 0;

				pMold->CoolPinBlow.Timer.IN = 0;
				pMold->CoolPinBlow.Step     = 0;
				break;

	 }/* end of switch */

	/* ----------------- cool pin blow  action limit --------------------  */
	 if(pMold->CoolPinBlow.Step > 100 && pMold->CoolPinBlow.Step < 900)
	 {
	 	if( 0 == pMold->Option.CoolPin && 1 == gMachineInfo.Auto)
	 	{
			pMold->CoolPinBlow.Step  = 900;
		}
	}
}/*end of function */
```

### Program Logical/process/coolblw2 (ANSIC, version 1.00.0) - cool blow 2

#### coolblow2.c
```c
/********************************************************************
 * COPYRIGHT --  B&R
 ********************************************************************
 * Program: coolblow
 * File: coolblow.c
 * Author: lijianjun
 * Created: March 06, 2013
 ********************************************************************
 * Implementation of program coolblow --- cooling blow control
 ********************************************************************/

#include <bur/plctypes.h>

#ifdef _DEFAULT_INCLUDES
#include <AsDefault.h>
#endif

/**************************************************************************************
                            Function Declarations
**************************************************************************************/

void CoolPin2Blow( Mold_typ * pMold);

/**************************************************************************************
     	        		I N I T U P  O F   T H E   T A S K
**************************************************************************************/
_INIT void init ( void )
 {
 	LMold.CoolPin2Blow.Step = 0;
 	RMold.CoolPin2Blow.Step = 0;
 } /* end of _INIT */

 /*************************************************************************************
        				C Y C L I C   P A R T   O F   T H E   T A S K
**************************************************************************************/

 _CYCLIC void cyclic ( void )
 {
	CoolPin2Blow(&LMold);
	CoolPin2Blow(&RMold);

	gMachineOut.LMold.CoolPin2Blow = LMold.ValveOut.CoolPin2Blow;
	gMachineOut.RMold.CoolPin2Blow = RMold.ValveOut.CoolPin2Blow;

 } /* end of _CYCLIC */

void CoolPin2Blow( Mold_typ * pMold)
{

	 switch ( pMold->CoolPin2Blow.Step )
     {
      		/*------------------ stop all the output ------------------*/
            case 0:
            	pMold->CoolPin2Blow.Out   	= 0;
            	pMold->ActInfo.CoolPin2Blow  = 0;
            	pMold->CoolPin2Blow.Timer.IN	= 0;
            	break;

      		/*------------------ CoolPin2 -------------------- */
            case 100:
            	if(pMold->Option.CoolPin2)
      			{
	            	if(pMold->TimeSet.CoolPin2BlowDelay != 0)
		      		{
	      				pMold->CoolPin2Blow.Timer.IN = 1;
						pMold->CoolPin2Blow.Timer.PT = pMold->TimeSet.CoolPin2BlowDelay;
	      				pMold->CoolPin2Blow.Step = 200;
	      			}
	      			else
	      			{
	      				pMold->CoolPin2Blow.Step = 300;
	      			}
	      		}
	      		else
	      		{
	      			pMold->CoolPin2Blow.Step = 900;
	      		}
            	break;
            case 200:
            	pMold->TimeDis.CoolPin2BlowDelay = pMold->CoolPin2Blow.Timer.ET;
            	if (1 == pMold->CoolPin2Blow.Timer.Q)
            	{
            		pMold->CoolPin2Blow.Timer.IN       = 0;
            //		pMold->TimeDis.CoolPin2BlowDelay = 0;
            		pMold->CoolPin2Blow.Step = 300;
            	}
            	break;
            case 300:
            	if(pMold->TimeSet.CoolPin2BlowTime != 0)
            	{
            		pMold->CoolPin2Blow.Timer.IN = 1;
					pMold->CoolPin2Blow.Timer.PT = pMold->TimeSet.CoolPin2BlowTime;
					pMold->CoolPin2Blow.Step = 400;
            	}
            	else
            	{
            		pMold->CoolPin2Blow.Step = 900;
            	}
            	break;
            case 400:
            	pMold->CoolPin2Blow.Out      = 1;
            	pMold->ActInfo.CoolPin2Blow  = 1;
            	pMold->ValveOut.CoolPin2Blow = 1;

            	pMold->TimeDis.CoolPin2BlowTime = pMold->CoolPin2Blow.Timer.ET;
            	if (1 == pMold->CoolPin2Blow.Timer.Q)
            	{
            		pMold->CoolPin2Blow.Out      = 0;
            		pMold->ActInfo.CoolPin2Blow  = 0;
            		pMold->ValveOut.CoolPin2Blow = 0;

            		pMold->CoolPin2Blow.Timer.IN = 0;
            	//	pMold->TimeDis.CoolPin2BlowTime = 0;

            		pMold->CoolPin2Blow.Step = 900;
            	}
            	break;
            case 900:
//			if (1==gMachineInfo.Auto)
//			{
//				if(pMold == &RMold)
//				{
//					RMold.Option.CoolPin2 = gMacOption.RCoolPin2;
//				}
//				else
//				{
//					LMold.Option.CoolPin2 = gMacOption.LCoolPin2;
//				}
//			}
            	pMold->CoolPin2Blow.Out      = 0;
            	pMold->ActInfo.CoolPin2Blow  = 0;
            	pMold->ValveOut.CoolPin2Blow = 0;

            	pMold->CoolPin2Blow.Timer.IN = 0;

            	pMold->CoolPin2Blow.Step = 3000;
            	break;

            case 3000:
            	break;

			case 5000:
				pMold->ActInfo.CoolPin2Blow  = 1;
				pMold->ValveOut.CoolPin2Blow = 1;

				break;

            case 20000:
            	pMold->CoolPin2Blow.Out      = 0;
            	pMold->ActInfo.CoolPin2Blow  = 0;
            	pMold->ValveOut.CoolPin2Blow = 0;

				pMold->CoolPin2Blow.Timer.IN = 0;
				pMold->CoolPin2Blow.Step    = 0;
				break;

			case 30000:
            	pMold->CoolPin2Blow.Out      = 0;
            	pMold->ActInfo.CoolPin2Blow  = 0;
            	pMold->ValveOut.CoolPin2Blow = 0;

				pMold->CoolPin2Blow.Timer.IN = 0;
				pMold->CoolPin2Blow.Step     = 0;
				break;

	 }/* end of switch */

	 if(pMold->CoolPin2Blow.Step > 100 && pMold->CoolPin2Blow.Step < 500)
	 {
	 	if(!pMold->Option.CoolPin2 && 1 == gMachineInfo.Auto)
	 	{
			pMold->CoolPin2Blow.Step  = 900;
		}
	}
}/*end of function */
```

### Program Logical/process/coolblw3 (ANSIC, version 1.00.0) - cool blow 3

#### coolblow3.c
```c
/********************************************************************
 * COPYRIGHT --  B&R
 ********************************************************************
 * Program: coolblow
 * File: coolblow.c
 * Author: lijianjun
 * Created: March 06, 2013
 ********************************************************************
 * Implementation of program coolblow --- cooling blow control
 ********************************************************************/

#include <bur/plctypes.h>

#ifdef _DEFAULT_INCLUDES
#include <AsDefault.h>
#endif

/**************************************************************************************
                            Function Declarations
**************************************************************************************/

void CoolPin3Blow( Mold_typ * pMold);

/**************************************************************************************
     	        		I N I T U P  O F   T H E   T A S K
**************************************************************************************/
_INIT void init ( void )
 {
 	LMold.CoolPin3Blow.Step = 0;
 	RMold.CoolPin3Blow.Step = 0;
 } /* end of _INIT */

 /*************************************************************************************
        				C Y C L I C   P A R T   O F   T H E   T A S K
**************************************************************************************/

 _CYCLIC void cyclic ( void )
 {
	CoolPin3Blow(&LMold);
	CoolPin3Blow(&RMold);

	gMachineOut.LMold.CoolPin3Blow = LMold.ValveOut.CoolPin3Blow;
	gMachineOut.RMold.CoolPin3Blow = RMold.ValveOut.CoolPin3Blow;

 } /* end of _CYCLIC */

void CoolPin3Blow( Mold_typ * pMold)
{

	 switch ( pMold->CoolPin3Blow.Step )
     {
      		/*------------------ stop all the output ------------------*/
            case 0:
            	pMold->CoolPin3Blow.Out   	= 0;
            	pMold->ActInfo.CoolPin3Blow  = 0;
            	pMold->CoolPin3Blow.Timer.IN	= 0;
            	break;

      		/*------------------ CoolPin3 -------------------- */
            case 100:
            	if(pMold->Option.CoolPin3)
      			{
	            	if(pMold->TimeSet.CoolPin3BlowDelay != 0)
		      		{
	      				pMold->CoolPin3Blow.Timer.IN = 1;
						pMold->CoolPin3Blow.Timer.PT = pMold->TimeSet.CoolPin3BlowDelay;
	      				pMold->CoolPin3Blow.Step = 200;
	      			}
	      			else
	      			{
	      				pMold->CoolPin3Blow.Step = 300;
	      			}
	      		}
	      		else
	      		{
	      			pMold->CoolPin3Blow.Step = 900;
	      		}
            	break;
            case 200:
            	pMold->TimeDis.CoolPin3BlowDelay = pMold->CoolPin3Blow.Timer.ET;
            	if (1 == pMold->CoolPin3Blow.Timer.Q)
            	{
            		pMold->CoolPin3Blow.Timer.IN       = 0;
            	//	pMold->TimeDis.CoolPin3BlowDelay = 0;
            		pMold->CoolPin3Blow.Step = 300;
            	}
            	break;
            case 300:
            	if(pMold->TimeSet.CoolPin3BlowTime != 0)
            	{
            		pMold->CoolPin3Blow.Timer.IN = 1;
					pMold->CoolPin3Blow.Timer.PT = pMold->TimeSet.CoolPin3BlowTime;
					pMold->CoolPin3Blow.Step = 400;
            	}
            	else
            	{
            		pMold->CoolPin3Blow.Step = 900;
            	}
            	break;
            case 400:
            	pMold->CoolPin3Blow.Out      = 1;
            	pMold->ActInfo.CoolPin3Blow  = 1;
            	pMold->ValveOut.CoolPin3Blow = 1;

            	pMold->TimeDis.CoolPin3BlowTime = pMold->CoolPin3Blow.Timer.ET;
            	if (1 == pMold->CoolPin3Blow.Timer.Q)
            	{
            		pMold->CoolPin3Blow.Out      = 0;
            		pMold->ActInfo.CoolPin3Blow  = 0;
            		pMold->ValveOut.CoolPin3Blow = 0;

            		pMold->CoolPin3Blow.Timer.IN = 0;
            	//	pMold->TimeDis.CoolPin3BlowTime = 0;

            		pMold->CoolPin3Blow.Step = 900;
            	}
            	break;
            case 900:
//			if (1==gMachineInfo.Auto)
//			{
//				if(pMold == &RMold)
//				{
//					RMold.Option.CoolPin3 = gMacOption.RCoolPin3;
//				}
//				else
//				{
//					LMold.Option.CoolPin3 = gMacOption.LCoolPin3;
//				}
//			}
            	pMold->CoolPin3Blow.Out      = 0;
            	pMold->ActInfo.CoolPin3Blow  = 0;
            	pMold->ValveOut.CoolPin3Blow = 0;

            	pMold->CoolPin3Blow.Timer.IN = 0;

            	pMold->CoolPin3Blow.Step = 3000;
            	break;

            case 3000:
            	break;

			case 5000:
				pMold->ActInfo.CoolPin3Blow  = 1;
				pMold->ValveOut.CoolPin3Blow = 1;

				break;

            case 20000:
            	pMold->CoolPin3Blow.Out      = 0;
            	pMold->ActInfo.CoolPin3Blow  = 0;
            	pMold->ValveOut.CoolPin3Blow = 0;

				pMold->CoolPin3Blow.Timer.IN = 0;
				pMold->CoolPin3Blow.Step    = 0;
				break;

			case 30000:
            	pMold->CoolPin3Blow.Out      = 0;
            	pMold->ActInfo.CoolPin3Blow  = 0;
            	pMold->ValveOut.CoolPin3Blow = 0;

				pMold->CoolPin3Blow.Timer.IN = 0;
				pMold->CoolPin3Blow.Step     = 0;
				break;

	 }/* end of switch */

	 if(pMold->CoolPin3Blow.Step > 100 && pMold->CoolPin3Blow.Step < 500)
	 {
	 	if(!pMold->Option.CoolPin3 && 1 == gMachineInfo.Auto)
	 	{
			pMold->CoolPin3Blow.Step  = 900;
		}
	}
}/*end of function */
```

### Program Logical/process/cutter (ANSIC, version 1.00.0) - cutter

#### cutter.c
```c
/********************************************************************
 * COPYRIGHT --  B&R
 ********************************************************************
 * Program: cutter
 * File: cutter.c
 * Author: lijianjun
 * Created: March 06, 2013
 ********************************************************************
 * Implementation of program cutter --- cutter control
 ********************************************************************/

#include <bur/plctypes.h>

#ifdef _DEFAULT_INCLUDES
#include <AsDefault.h>
#endif

#include "edge.h"

/**************************************************************************************
                            Function Declarations
**************************************************************************************/

void Cutter( Mold_typ * pMold);

/**************************************************************************************
     	        		I N I T U P  O F   T H E   T A S K
**************************************************************************************/
_INIT void init ( void )
 {
 	LMold.Cutter.Step = 0;
 	RMold.Cutter.Step = 0;
 } /* end of _INIT */

 /*************************************************************************************
        				C Y C L I C   P A R T   O F   T H E   T A S K
**************************************************************************************/

 _CYCLIC void cyclic ( void )
 {

	Cutter(&LMold);
	Cutter(&RMold);

//	if(1 == gMachineInfo.Auto)
//	{
//		if( 1 == LMold.Option.CutterMode)	/*  双向切刀 */
//		{
//			if(0 == LMold.ValveOut.Cutter && 0 == RMold.ValveOut.Cutter)
//			{
//				gMachineOut.CutterFw = 0;
//				gMachineOut.CutterBw = 0;
//			}
//			else if(1 == LMold.ValveOut.Cutter || 1 == RMold.ValveOut.Cutter)
//			{
//				gMachineOut.CutterFw = 1;
//				gMachineOut.CutterBw = 0;
//			}
//			else
//			{
//				gMachineOut.CutterFw = 0;
//				gMachineOut.CutterBw = 1;
//			}
//		}
//		else								/*  单向切刀 */
//		{
//			if (EDGEPOS(LMold.ValveOut.Cutter ,Cutter_L_P) || EDGEPOS(RMold.ValveOut.Cutter ,Cutter_R_P))
//			{
//				if(0 == gMachineOut.CutterBw)
//				{
//					gMachineOut.CutterFw = !gMachineOut.CutterFw;
//				}
//
//				if(0 == gMachineOut.CutterFw)
//				{
//					gMachineOut.CutterBw = !gMachineOut.CutterBw;
//					if(0 == gMachineOut.CutterBw)gMachineOut.CutterFw = ! gMachineOut.CutterFw;
//				}
//			}
//		}
//	}
//	else
//	{
//		if(0 == LMold.ValveOut.Cutter && 0 == RMold.ValveOut.Cutter)
//		{
//			gMachineOut.CutterFw = 0;
//			gMachineOut.CutterBw = 0;
//		}
//		else if(1 == LMold.ValveOut.Cutter || 1 == RMold.ValveOut.Cutter)
//		{
//			gMachineOut.CutterFw = 1;
//			gMachineOut.CutterBw = 0;
//		}
//		else
//		{
//			gMachineOut.CutterFw = 0;
//			gMachineOut.CutterBw = 1;
//		}
//	}

//	Cutter_L_P = LMold.ValveOut.Cutter;
//	Cutter_R_P = RMold.ValveOut.Cutter;

	gMachineOut.CutterFw = LMold.ValveOut.Cutter | RMold.ValveOut.Cutter;
 } /* end of _CYCLIC */

void Cutter( Mold_typ * pMold)
{
	 switch ( pMold->Cutter.Step )
     {
      		/*------------------ stop all the output ------------------*/
            case 0:
//            	pMold->ValveOut.Cutter  	   = 0;
//            	pMold->ActInfo.Cutter  = 0;

            	pMold->Cutter.Timer.IN	= 0;
            	break;

      		/*------------------ Cutter course -------------------- */
      		case 100: /* close delay*/
			if ( pMold->Option.Cutter)
			{
				if(pMold->TimeSet.CutterDelay != 0)
				{
					pMold->Cutter.Timer.IN = 1;
					pMold->Cutter.Timer.PT = pMold->TimeSet.CutterDelay;
					pMold->Cutter.Step 	   = 200;
				}
				else
				{
					pMold->Cutter.Step = 300;
				}
			}
			else
			{
				pMold->Cutter.Step = 3000;
			}

             	break;

            case 200: /* delay ok */
            	pMold->TimeDis.CutterDelay = pMold->Cutter.Timer.ET;
            	if (1 == pMold->Cutter.Timer.Q)
            	{
            		pMold->Cutter.Timer.IN     = 0;
            	//	pMold->TimeDis.CutterDelay = 0;
            		pMold->Cutter.Step = 300;
            	}
            	break;

            case 300:/*Determine Cutter mode , if double cutter goes to 400, single cutter goes to 1100*/
					/*   涨气启动   */
//				RMold.SupportAir.Step = 100;
				if(1 == gMachineInfo.Auto)
				{
//						if(RMold.SupportAir.Step == 0)RMold.SupportAir.Step = 100;

					if(1 == RMold.Option.Enable && 1 == LMold.Option.Enable)
					{
						if(pMold == &RMold)
						{
							LMold.OnceSupport  = 1;
						}
						else
						{
							RMold.OnceSupport  = 1;
						}
					}
					else
					{
						pMold->OnceSupport  = 1;
					}
				}

            	if( 1 == pMold->Option.CutterMode)/*Double Cutter*/
            	{
					if( 0 ==  pMold->ValveOut.Cutter)
					{
						if( SUPPORTAIR_MODE_STANDARD == gMachineFix.MoldR.SupportAir.eSupportAirMode)
						{
							pMold->SupportAir.Step = 100;// air support， only for double cutter
						}

						if(pMold->TimeSet.CutterTime != 0)
						{
							pMold->Cutter.Timer.IN = 1;
							pMold->Cutter.Timer.PT = pMold->TimeSet.CutterTime;
							pMold->Cutter.Step = 400;
						}
						else
						{
							/*   cutter time gAlarm   */
							pMold->Cutter.Step = 450;
						}

					}
					else /*If cutter is retain on Fw position , then do Single Cutter again to go back Bw Position*/
					{
						pMold->Cutter.Step = 1100;
					}

	            }
	            else/*Single Cutter*/
	            {
	            	pMold->Cutter.Step = 1100;
	            }
            	break;

            case 400:/*Double cutter, move forward until time expired*/
            	pMold->ActInfo.Cutter = 1;
				pMold->ValveOut.Cutter  = 1;

            	pMold->TimeDis.CutterTime = pMold->Cutter.Timer.ET;
            	if (1 == pMold->Cutter.Timer.Q)
            	{
            		pMold->Cutter.Timer.IN    = 0;
            //		pMold->TimeDis.CutterTime = 0;
					pMold->Cutter.Step = 450;/*Change to case 450*/
            	}
            	break;

			case 450:/*Time expire or no cutter time setting*/
				pMold->ValveOut.Cutter = 0;
				pMold->ActInfo.Cutter  = 0;

				pMold->Cutter.Step 	  = 3000;
			break;

            case 500:/*Current no used case*/
            	pMold->Cutter.Timer.IN = 1;
					pMold->Cutter.Timer.PT = pMold->TimeSet.CutterBwTime;
					pMold->Cutter.Step = 600;
            	break;

            case 600:/*Current no used case*/
            	pMold->ValveOut.Cutter     = 2;
            	pMold->ActInfo.Cutter = 1;

            	pMold->TimeDis.CutterBwTime = pMold->Cutter.Timer.ET;
            	if (1 == pMold->Cutter.Timer.Q)
            	{
            		pMold->Cutter.Timer.IN      = 0;
            	//	pMold->TimeDis.CutterBwTime = 0;
            		pMold->Cutter.Step = 700;
            	}
				break;

            case 700:/*Current no used case*/
            	pMold->ValveOut.Cutter = 0;
            	pMold->ActInfo.Cutter  = 0;

				pMold->Cutter.Step = 800;
            	break;

            case 800:/*Current no used case*/
            	pMold->ValveOut.Cutter     = 0;
            	pMold->ActInfo.Cutter = 0;

            	pMold->Cutter.Step = 3000;
            	break;

            case 1100:/*Single cutter , inverse output*/
            	pMold->ValveOut.Cutter = !pMold->ValveOut.Cutter;/*Albert*/
            	pMold->ActInfo.Cutter = pMold->ValveOut.Cutter;
            	pMold->Cutter.Step = 3000;
            	break;

            case 1200:/*Current no used case*/
            	pMold->Cutter.Step = 1300;
            	break;

            case 1300:/*Current no used case*/
               	pMold->ValveOut.Cutter     = 0;
            	pMold->ActInfo.Cutter = 0;

            	pMold->Cutter.Step = 3000;
            	break;

            case 3000:
            	break;

			case 5000:
				pMold->ValveOut.Cutter     = 1;
				pMold->ActInfo.Cutter = 1;
				break;

            /*--------------- Manual action stop -----------------*/
            case 20000:
				if(pMold->Option.CutterMode)/*Albert Double cutter*/
				{
					pMold->ValveOut.Cutter      = 0;
				}

					pMold->Cutter.Timer.IN = 0;

				//	pMold->TimeDis.CutterTime  = 0;
				//	pMold->TimeDis.CutterDelay = 0;

					pMold->ActInfo.Cutter  = 0;
					pMold->Cutter.Step 	   = 0;
					break;

			/*--------------- Instance stop -----------------*/
			case 30000:
				if(pMold->Option.CutterMode)/*Albert Double Cutter*/
				{
					pMold->ValveOut.Cutter      = 0;
				}
				pMold->Cutter.Timer.IN = 0;

			//	pMold->TimeDis.CutterTime  = 0;
			//	pMold->TimeDis.CutterDelay = 0;

				pMold->ActInfo.Cutter  = 0;
				pMold->Cutter.Step     = 0;
				break;

	 }/* end of switch */
}/*end of function */
```

#### cutter.var
```iecst
VAR
	Cutter_R_P	:USINT;
	Cutter_L_P	:USINT;
END_VAR
```

- edge.h (reference to Logical/GlobalIncludes/edge.h)

### Program Logical/process/sensor (ANSIC, version 1.00.0) - sensor up / down

#### sensor.c
```c
/********************************************************************
 * COPYRIGHT --  B&R China
 ********************************************************************
 * Program: Tonnage
 * File: Tonnage.c
 * Author: lijianjun
 * Created: March 06, 2013
 ********************************************************************
 * Implementation of program Tonnage --- mold Tonnage
 ********************************************************************/

#include <bur/plctypes.h>

#ifdef _DEFAULT_INCLUDES
	#include <AsDefault.h>
#endif

/**************************************************************************************
                            Function Declarations
**************************************************************************************/

void Sensor( Mold_typ * pMold,Robot_Para_typ * pRobotPara);

/**************************************************************************************
     	        		I N I T U P  O F   T H E   T A S K
**************************************************************************************/
_INIT void init ( void )
 {
	RTInfo_Task.enable = 1;
	RTInfo(&RTInfo_Task);

	tTask = RTInfo_Task.cycle_time/1000.0/1000.0;		/*  from us ---> s  */

 	LMold.Sensor.Step = 30000;
 	RMold.Sensor.Step = 30000;
 } /* end of _INIT */

 /*************************************************************************************
        				C Y C L I C   P A R T   O F   T H E   T A S K
**************************************************************************************/

 _CYCLIC void cyclic ( void )
 {
	LMold.TransDIn.SensorUp = gMachineIn.LMold.SensorUp = 1;
	RMold.TransDIn.SensorUp = gMachineIn.RMold.SensorUp = 1;

	Sensor(&LMold,&gMachinePara.MoldL.Robot);
	Sensor(&RMold,&gMachinePara.MoldR.Robot);

 } /* end of _CYCLIC */

void Sensor( Mold_typ * pMold,Robot_Para_typ * pRobotPara)
{
	pMold->Sensor.UpDn.CalOK = pMold->Sensor.UpDn.HomingOk = 1;

	pRobotPara->ParaUpDn.sSensorBottle = 0.0;
	pRobotPara->ParaUpDn.sSensorWaste  = 0.0;

	pMold->Sensor.UpDn.mmAs = 0.0;

	if(pMold->TimeSet.SensorUpAlarmTime < 10)pMold->TimeSet.SensorUpAlarmTime = 1000;
	if(pMold->TimeSet.SensorDnAlarmTime < 10)pMold->TimeSet.SensorDnAlarmTime = 1000;

	if((1 == pMold->Sensor.UpDn.HomingOk) &&  (1 == pMold->TransDIn.SensorUp) &&
		(pMold->Sensor.UpDn.mmAs > -0.2  ) && (pMold->Sensor.UpDn.mmAs < 0.2))
	{
		pMold->Sensor.ZeroPos = 1;
	}
	else
	{
		pMold->Sensor.ZeroPos = 0;
	}

	if((1 == pMold->Sensor.UpDn.HomingOk) &&
		(pMold->Sensor.UpDn.mmAs > pRobotPara->ParaUpDn.sSensorBottle - 0.2) &&
		(pMold->Sensor.UpDn.mmAs < pRobotPara->ParaUpDn.sSensorBottle + 0.2    ))
	{
		pMold->Sensor.BottlePos = 1;
	}
	else
	{
		pMold->Sensor.BottlePos = 0;
	}

	if((1 == pMold->Sensor.UpDn.HomingOk) &&
		(pMold->Sensor.UpDn.mmAs > pRobotPara->ParaUpDn.sSensorWaste - 0.2) &&
		(pMold->Sensor.UpDn.mmAs < pRobotPara->ParaUpDn.sSensorWaste + 0.2    ))
	{
		pMold->Sensor.WastePos = 1;
	}
	else
	{
		pMold->Sensor.WastePos = 0;
	}

	switch ( pMold->Sensor.Step )
   {
   		/*------------------ stop all the output ------------------*/
         case 0:
				 pMold->Sensor.UpDn.v_set = 0;
         	 pMold->Sensor.Timer.IN	= 0;
         	break;

   		/*------------------ Sensor down -------------------- */
   		case 100: 	/* delay */
				if(1 == pMold->Option.HookPin)
				{
					pMold->Sensor.Timer.IN = 1;
					pMold->Sensor.Timer.PT = 1;
					pMold->Sensor.Step = 200;
				}
				else
				{
					pMold->Sensor.Step = 3000;
				}
            break;

         case 200: 	/* Sensoring delay */
            if (1 == pMold->Sensor.Timer.Q)
            {
               pMold->Sensor.Timer.IN = 0;
               pMold->Sensor.Step = 300;
            }
            break;

         case 300: 	/* scan Sensor bottle */
				pMold->Sensor.LimitTimer.IN = 1;
				pMold->Sensor.LimitTimer.PT = pMold->TimeSet.SensorDnAlarmTime;

				pMold->Sensor.UpDn.s_set = pRobotPara->ParaUpDn.sSensorBottle;
				pMold->Sensor.UpDn.MoveAbsolute = 1;
				pMold->Sensor.Step = 400;
            break;

         case 400:
				pMold->TimeDis.SensorDnAlarmTime = pMold->Sensor.LimitTimer.ET;

				if(1 == pMold->Sensor.LimitTimer.Q)
				{
					pMold->Sensor.LimitTimer.IN = 0;
					pMold->Sensor.Step = 40000;
				}

				if(pMold->Sensor.UpDn.mmAs > pRobotPara->ParaUpDn.sSensorBottle - 0.02 && pMold->Sensor.UpDn.mmAs < pRobotPara->ParaUpDn.sSensorBottle + 0.02)
				{
					pMold->Sensor.LimitTimer.IN = 0;
					pMold->Sensor.Step = 3000;
				}

            break;

			/*------------------ Sensor down -------------------- */
			case 1100: 	/* delay */
				if(1 == pMold->Option.HookPin)
				{
					pMold->Sensor.Timer.IN = 1;
					pMold->Sensor.Timer.PT = 1;
					pMold->Sensor.Step = 1200;
				}
				else
				{
					pMold->Sensor.Step = 3000;
				}
				break;

			case 1200: 	/* Sensoring delay */
				if (1 == pMold->Sensor.Timer.Q)
				{
					pMold->Sensor.Timer.IN = 0;
					pMold->Sensor.Step = 1300;
				}
				break;

			case 1300: 	/* scan Sensor bottle */
				pMold->Sensor.LimitTimer.IN = 1;
				pMold->Sensor.LimitTimer.PT = pMold->TimeSet.SensorDnAlarmTime;

				pMold->Sensor.UpDn.s_set = pRobotPara->ParaUpDn.sSensorWaste;
				pMold->Sensor.UpDn.MoveAbsolute = 1;
				pMold->Sensor.Step = 1400;
				break;

			case 1400:
				pMold->TimeDis.SensorDnAlarmTime = pMold->Sensor.LimitTimer.ET;
				if(1 == pMold->Sensor.LimitTimer.Q)
				{
					pMold->Sensor.LimitTimer.IN = 0;
					pMold->Sensor.Step = 40000;
				}

				if(pMold->Sensor.UpDn.mmAs > pRobotPara->ParaUpDn.sSensorBottle - 0.02 && pMold->Sensor.UpDn.mmAs < pRobotPara->ParaUpDn.sSensorBottle + 0.02)
				{
					pMold->Sensor.LimitTimer.IN = 0;
					pMold->Sensor.Step = 3000;
				}
				break;

			case 3000:
				break;

			/*  sensor calibration down    */
			case 5000:
				if(0 == pMold->Sensor.UpDn.BwHWSwitch)
				{
					pMold->Sensor.UpDn.v_set = pRobotPara->ParaUpDn.vSensorHome;
				}

				if(1 == pMold->Sensor.UpDn.BwHWSwitch)
				{
					pMold->HwAlarm.SensorDnHWSwitch = 1;
					pMold->BlowPin.Step 	= 25000;
				}
				break;

			/*  sensor up   */
         case 10100:
				if(1 == pMold->Option.HookPin)
				{
					pMold->Sensor.Timer.IN = 1;
					pMold->Sensor.Timer.PT = 1;
					pMold->Sensor.Step = 10200;
				}
				else
				{
					pMold->Sensor.Step = 13000;
				}
            break;

         case 10200:
				if (1 == pMold->Sensor.Timer.Q)
				{
					pMold->Sensor.Timer.IN = 0;
					pMold->Sensor.Step = 10300;
				}
            break;

         case 10300:
				pMold->Sensor.LimitTimer.IN = 1;
				pMold->Sensor.LimitTimer.PT = pMold->TimeSet.SensorUpAlarmTime;

				pMold->Sensor.UpDn.s_set = 0;
				pMold->Sensor.UpDn.MoveAbsolute = 1;
				pMold->Sensor.Step = 10400;
            break;

         case 10400:
				pMold->TimeDis.SensorUpAlarmTime = pMold->Sensor.LimitTimer.ET;
				if(1 == pMold->Sensor.LimitTimer.Q)
				{
					pMold->Sensor.LimitTimer.IN = 0;
					pMold->Sensor.Step = 40000;
				}

				if(pMold->Sensor.UpDn.mmAs > -0.02 && pMold->Sensor.UpDn.mmAs < 0.02)
				{
					pMold->Sensor.LimitTimer.IN = 0;
					pMold->Sensor.Step = 13000;
				}
            break;

         case 13000:
            break;

			/*  Sensor calibration up    */
			case 15000:
				if(0 == pMold->Sensor.UpDn.FwHWSwitch)
				{
					pMold->Sensor.UpDn.v_set = -pRobotPara->ParaUpDn.vSensorHome;
				}

				if(1 == pMold->Sensor.UpDn.BwHWSwitch)
				{
					pMold->HwAlarm.SensorUpHWSwitch = 1;
					pMold->BlowPin.Step = 25000;
				}
				break;

        /*--------------- Manual action stop -----------------*/
         case 20000:
				pMold->Sensor.UpDn.MoveAbsolute = 0;
				pMold->Sensor.UpDn.Stop = 1;
				pMold->Sensor.Timer.IN = 0;
         	pMold->Sensor.Step = 0;
            break;

			case 25000:
				pMold->Sensor.vRamp.Ts = tTask;
				pMold->Sensor.vRamp.Once = 0;
				pMold->Sensor.vRamp.Set = pMold->Sensor.UpDn.v_set;
				pMold->Sensor.vRamp.Accel = 1000;

				/* call profile function */
				HydSCurveRamp(&pMold->Sensor.vRamp);
				pMold->Sensor.UpDn.v_set = pMold->Sensor.vRamp.Out;

				pMold->Sensor.Step = 26000;
				break;

			case 26000:
				pMold->Sensor.vRamp.Set = 0;
				pMold->Sensor.vRamp.Accel = 1000;

				/* call profile function */
				HydSCurveRamp(&pMold->Sensor.vRamp);
				pMold->Sensor.UpDn.v_set = pMold->Sensor.vRamp.Out;

				if(pMold->Sensor.UpDn.v_set < 0.1 && pMold->Sensor.UpDn.v_set > -0.1)
				{
					pMold->Sensor.UpDn.v_set = 0;
					pMold->Sensor.Step = 0;
				}
				break;
			/*--------------- Instance stop -----------------*/
			case 30000:
				pMold->Sensor.UpDn.v_set = 0;
				pMold->Sensor.UpDn.MoveJogPos = 0;
				pMold->Sensor.UpDn.MoveJogNeg = 0;
           	pMold->Sensor.Timer.IN = 0;
           	pMold->Sensor.Step = 0;
            break;

			/*--------------- Instance stop -----------------*/
			case 40000:
				pMold->Sensor.UpDn.Stop = 1;
				pMold->Sensor.UpDn.v_set = 0;
				pMold->Sensor.Timer.IN = 0;
				pMold->Sensor.Step = 0;
				break;
	}/* end of switch */
}/*end of function */
```

#### sensor.var
```iecst
VAR
	tTask : REAL := 0.0;
	RTInfo_Task : RTInfo := (0);
END_VAR
```

### Program Logical/process/robot (ANSIC, version 1.00.0) - robot
